PROGRAM MAPPING_in
VAR CONSTANT
{IF defined (AXIS_MAP)}
  {info 'MAPPING_in - ACTIVE'}
  bBypassMapping    : BOOL  := FALSE;
{ELSE}
  bBypassMapping    : BOOL  := TRUE;
{END_IF}
END_VAR
VAR
{IF defined (AXIS_MAP)}
  AxisCTrl          : U_AXIS_CTRL;
  AxisMoveData      : U_AXIS_MOVE_DATA;
  AxisMotionOptions : U_AXIS_MOTION_OPTIONS;

  AxisGearInData    : U_AXIS_GEAR_IN;
  AxisHoming        : U_AXIS_HOMING;
  AxisParameterWrt  : U_AXIS_NC_PARAMETER_WRT;
  
{ELSE}
  AxisCTrl          : BYTE;
  AxisMoveData      : BYTE;
  AxisMotionOptions : BYTE;

  AxisGearInData    : BYTE;
  AxisHoming        : BYTE;
  AxisParameterWrt  : BYTE;
{END_IF}

  szAxisPara,
  szAxisHoming,
  szAxisGearData,
  szAxisMotionOptions,
  szAxisMoveData,
  szAxisCtrl        : ARRAY[1..2] OF UDINT;


END_VAR


szAxisCtrl[1]           := SIZEOF(AxisCTrl);
szAxisCtrl[2]           := SIZEOF(GVL_AXIS.Ctrl);

szAxisMoveData [1]      := SIZEOF(AxisMoveData);
szAxisMoveData [2]      := SIZEOF(GVL_AXIS.Data);

szAxisMotionOptions [1] := SIZEOF(AxisMotionOptions);
szAxisMotionOptions [2] := SIZEOF(GVL_AXIS.MotionOptions);

szAxisGearData [1]      := SIZEOF(AxisGearInData);
szAxisGearData [2]      := SIZEOF(GVL_AXIS.GearInParameter);

szAxisHoming [1]        := SIZEOF(AxisHoming);
szAxisHoming [2]        := SIZEOF(GVL_AXIS.HomeParameter);

szAxisPara [1]          := SIZEOF(AxisParameterWrt);
szAxisPara [2]          := SIZEOF(GVL_AXIS.NcParameterWrt);



IF bBypassMapping 
THEN 
  RETURN; 
END_IF


memcpy(ADR(GVL_AXIS.Ctrl),            ADR(AxisCtrl),           SIZEOF(AxisCTrl));
memcpy(ADR(GVL_AXIS.Data),            ADR(AxisMoveData),       SIZEOF(AxisMoveData));
memcpy(ADR(GVL_AXIS.MotionOptions),   ADR(AxisMotionOptions),  SIZEOF(AxisMotionOptions));

memcpy(ADR(GVL_AXIS.GearInParameter), ADR(AxisGearInData),     SIZEOF(AxisGearInData));
memcpy(ADR(GVL_AXIS.HomeParameter),   ADR(AxisHoming),         SIZEOF(AxisHoming));
memcpy(ADR(GVL_AXIS.NcParameterWrt),  ADR(AxisParameterWrt),   SIZEOF(AxisParameterWrt));

END_PROGRAM

(* stored: Version 1.1.0.1, ProductVersion 3.1.4024.12
   POU MAPPING_in: Id {e84de69b-ba26-07ad-1592-7be68e226b51}, SpecialFunc None *)
